(* PLC project RACK2537.project, Inovance company InoProShop(V1.8.1.3) InoProShop(V1.8.1.3) *)
(* stored: creationDateTime 2025-03-07T16:08:32.1498014, modificationDateTime 2025-03-07T16:07:54.7010798 *)

PROGRAM PLC_PRG
  VAR
    X_EN : BOOL;
    X_FWK : BOOL;
    X_FWKS : BOOL;
    X_TYYXH : BOOL;
    X_LYYS : BOOL;
    X_LYYXH : BOOL;
    X_LDXH : BOOL;
    X_LRYYXH : BOOL;
    Y_ENO : BOOL;
    FWZ : BOOL;
    X_FWWC : BOOL;
    Y_TCYY : BOOL;
    Y_LCYY : BOOL;
    Y_LJCYY : BOOL;
    Y_LJCDW : BOOL;
    Y_LRCYY : BOOL;
    XY_LGJ : BOOL;
    FWBZ : INT;
  END_VAR
  VAR  (* added by the conversion: wires and edge detectors of the diagram *)
    _EQ21_ENO : BOOL;
    _EQ21_OUT : BOOL;
    _EQ34_ENO : BOOL;
    _EQ34_OUT : BOOL;
    _EQ42_ENO : BOOL;
    _EQ42_OUT : BOOL;
    _EQ63_ENO : BOOL;
    _EQ63_OUT : BOOL;
    _EQ73_ENO : BOOL;
    _EQ73_OUT : BOOL;
  END_VAR

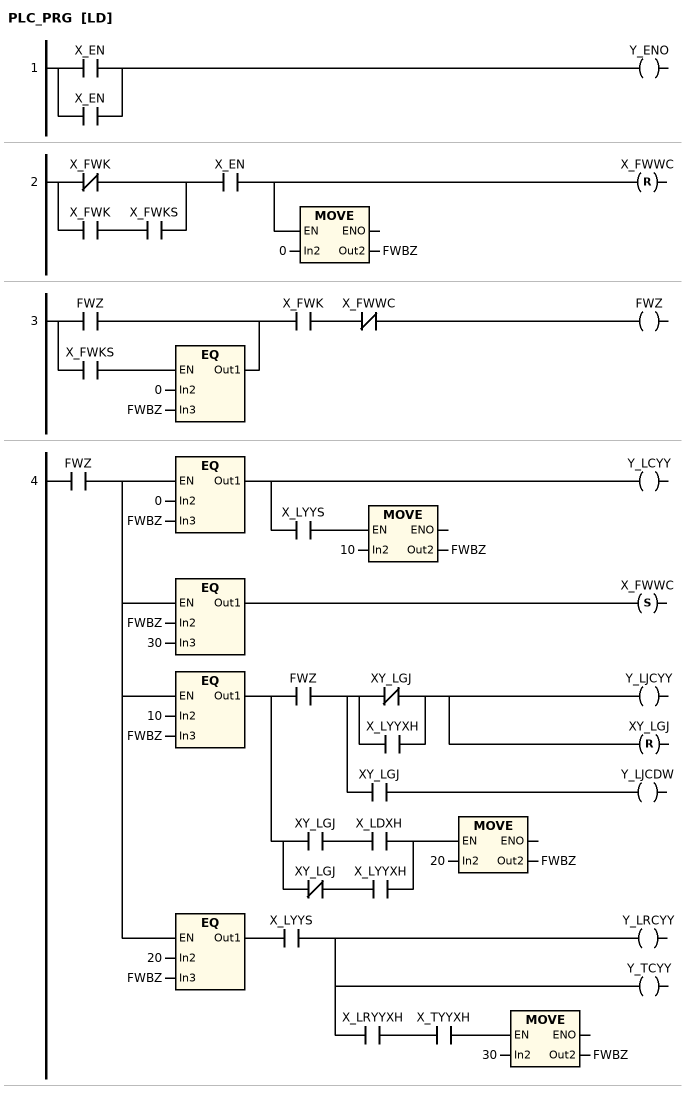
(* LD diagram, written out as Structured Text *)
(* 网络注释 *)

Y_ENO := X_EN;
(* 网络注释 *)

IF (NOT X_FWK OR X_FWK AND X_FWKS) AND X_EN THEN X_FWWC := FALSE; END_IF;
IF (NOT X_FWK OR X_FWK AND X_FWKS) AND X_EN THEN FWBZ := 0; END_IF;
(* 网络注释 *)

_EQ21_OUT := EQ(EN := X_FWKS, IN1 := 0, IN2 := FWBZ, ENO => _EQ21_ENO);
FWZ := (_EQ21_OUT OR FWZ) AND X_FWK AND NOT X_FWWC;
(* 网络注释 *)

_EQ34_OUT := EQ(EN := FWZ, IN1 := 0, IN2 := FWBZ, ENO => _EQ34_ENO);
Y_LCYY := _EQ34_OUT;
IF _EQ34_OUT AND X_LYYS THEN FWBZ := 10; END_IF;
_EQ42_OUT := EQ(EN := FWZ, IN1 := 10, IN2 := FWBZ, ENO => _EQ42_ENO);
Y_LJCYY := _EQ42_OUT AND FWZ AND (NOT XY_LGJ OR X_LYYXH);
IF _EQ42_OUT AND FWZ AND (NOT XY_LGJ OR X_LYYXH) THEN XY_LGJ := FALSE; END_IF;
Y_LJCDW := _EQ42_OUT AND FWZ AND XY_LGJ;
IF _EQ42_OUT AND (XY_LGJ AND X_LDXH OR NOT XY_LGJ AND X_LYYXH) THEN FWBZ := 20; END_IF;
_EQ63_OUT := EQ(EN := FWZ, IN1 := 20, IN2 := FWBZ, ENO => _EQ63_ENO);
Y_LRCYY := _EQ63_OUT AND X_LYYS;
Y_TCYY := _EQ63_OUT AND X_LYYS;
IF _EQ63_OUT AND X_LYYS AND X_LRYYXH AND X_TYYXH THEN FWBZ := 30; END_IF;
_EQ73_OUT := EQ(EN := FWZ, IN1 := FWBZ, IN2 := 30, ENO => _EQ73_ENO);
IF _EQ73_OUT THEN X_FWWC := TRUE; END_IF;
END_PROGRAM
